FUNCTION_BLOCK GREENTIMER (* Define minimum green times *)
  (* Standard: 61499-1-A.18; Classification: Event-driven blocks; Function: Up-counter *)
  (* Version 0.5, 2018-08-20, JHC, Holobloc Inc, Added ECC documentation. *)
  (* Version 0.4, 2018-08-11, JHC, Holobloc Inc, Added CV comment. *)
  (* Version 0.3, 2009-11-16, JHC, Holobloc Inc, Updated for 61499-1 Ed2. *)
  (* Version 0.2, 2006-09-07, JHC, Holobloc Inc, Changed package to fb.rt.events. *)
  (* Version 0.1, 2001-04-27, JHC, Rockwell Automation, XML version *)
  (* Version 0.0, 1999-01-22, JHC, Rockwell Automation, SRC version *)
  (* Compiler header: package fb.rt.events; *)
  (* Compiler Java Sun JDK 1.7.0 *)
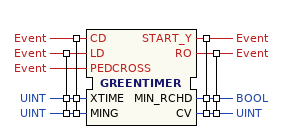
  EVENT_INPUT
    CD WITH XTIME, MING; (* Count Down *)
    LD WITH XTIME, MING; (* Reset *)
    PEDCROSS;
  END_EVENT
  EVENT_OUTPUT
    START_Y WITH MIN_RCHD, CV; (* Count Up Output Event *)
    RO WITH MIN_RCHD, CV; (* Reset Output Event *)
  END_EVENT
  VAR_INPUT
    XTIME : UINT; (* LImit Value *)
    MING : UINT;
  END_VAR
  VAR_OUTPUT
    MIN_RCHD : BOOL; (* CV >= PV *)
    CV : UINT; (* Current Value *)
  END_VAR
  VAR
    YELLOWSET : BOOL;
    PEDWANTSTOCROSS : BOOL;
  END_VAR
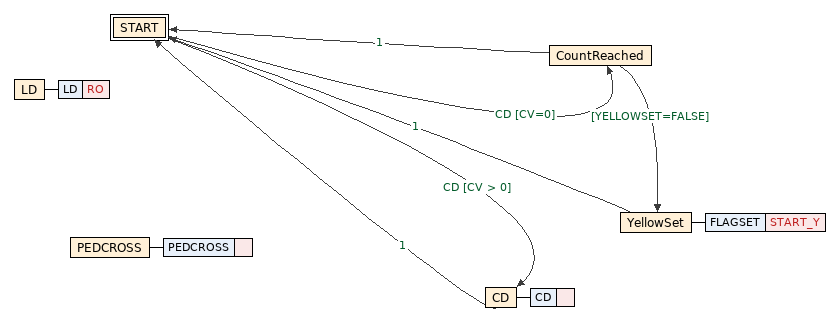
  EC_STATES
    START; (* Initial State *)
    CD : CD; (* Count Up *)
    LD : LD -> RO; (* Service R (Reset) Event *)
    CountReached;
    YellowSet : FLAGSET -> START_Y;
    PEDCROSS : PEDCROSS;
  END_STATES
  EC_TRANSITIONS
    CD TO START := 1;
    START TO CountReached := CD [CV=0];
    START TO CD := CD [CV > 0];
    CountReached TO YellowSet := [YELLOWSET=FALSE];
    YellowSet TO START := 1;
    CountReached TO START := 1;
  END_TRANSITIONS
  ALGORITHM CD IN ST: (* Count Up *)
CV := CV - 1;
  END_ALGORITHM
  ALGORITHM LD IN ST: (* Reset *)
CV := XTIME;
MIN_RCHD := FALSE;
YELLOWSET := FALSE;
  END_ALGORITHM
  ALGORITHM FLAGSET IN ST:
IF CV = 0 THEN
	YELLOWSET := TRUE;
END_IF;
  END_ALGORITHM
  ALGORITHM PEDCROSS IN ST:
CV := 0;
YELLOWSET := TRUE;
  END_ALGORITHM
END_FUNCTION_BLOCK
